Staubli VAL3: mnuMoveTargPnt.pgx

program mnuMoveTargPnt()
  local bool LbBackup
  local bool LbIsInRange
  local bool LbTestLocResult
  local joint LjHere
  local joint LjTarget
  local point LpMoveTarget
  local num nKey
begin
  //header begin
  // PROGRAM mnuMoveTargPnt()
  //
  // runs the menu to query for user to select and move to
  // Target Point
  //
  // incoming parms:  none
  // outgoing parms:  none
  // called from:  pgm mnuMotionMenu()
  //
  //  initial release KN
  //header end
  //
  // start continuous loop, end by menu command or teach pendant command
  // on user command, jump to other subroutines for action
  //
  // init booleans for menu control
  LbBackup=false
  bWorldFrameView=true
  //
  do
    //nIdxMoveTargPt=281
    call displayMessage2(nIdxMoveTargPt,nKey)
    // verify selection
    switch nKey
      // ESC key aborts & returns immediately
      case 255
        return
      break
      // Move to Target Point, F1 to change Target Frame number 1 or 2
      case 271
        nIPNumber=nIPNumber+1
        if nIPNumber==2
          nIPNumber=0
        endIf
      break
      // Move to Target Point, F2 to increment point number 0-19 in selected frame 0-1
      case 272
        if nIPNumber==0
          nIP1Number=nIP1Number+1
          if nIP1Number==20
            nIP1Number=0
          endIf
        else
          nIP2Number=nIP2Number+1
          if nIP2Number==20
            nIP2Number=0
          endIf
        endIf
      break
      // menu Move To Target Point, F5 to ADJUST RX/RY/RZ values of Target Point
      case 275
        call mnuAdjTargetPnt()
      break
      //  Move to Target Point, F6 to MOVE to currently selected IP & TP
      case 276
        // test if move to Target Point is possible
        // set up dummy loc at current location & configuration
        LjHere=jPark
        // test desired Target Point for validity
        if nIPNumber==0


          logMsg("x  "+toString(".6",tSensorTool.trsf.x))
          logMsg("y  "+toString(".6",tSensorTool.trsf.y))
          logMsg("z  "+toString(".6",tSensorTool.trsf.z))
          logMsg("rx "+toString(".6",tSensorTool.trsf.rx))
          logMsg("ry "+toString(".6",tSensorTool.trsf.ry))
          logMsg("rz "+toString(".6",tSensorTool.trsf.rz))

          logMsg("x  "+toString(".6",pIP1Point[nIP1Number].trsf.x))
          logMsg("y  "+toString(".6",pIP1Point[nIP1Number].trsf.y))
          logMsg("z  "+toString(".6",pIP1Point[nIP1Number].trsf.z))
          logMsg("rx "+toString(".6",pIP1Point[nIP1Number].trsf.rx))
          logMsg("ry "+toString(".6",pIP1Point[nIP1Number].trsf.ry))
          logMsg("rz "+toString(".6",pIP1Point[nIP1Number].trsf.rz))


          LbTestLocResult=pointToJoint(tSensorTool,LjHere,pIP1Point[nIP1Number],LjTarget)
        else
          LbTestLocResult=pointToJoint(tSensorTool,LjHere,pIP2Point[nIP2Number],LjTarget)
        endIf
        // issue error if not valid or if cannot be reached, otherwise commence move
        if LbTestLocResult==false
          LbBackup=true
          popUpMsg("IMPOSSIBLE MOVE:  Unable to reach Target Point in current arm configuration...Press OK")
          //call movTargetPoint()
        else
          LbIsInRange=isInRange(LjTarget)
          if LbIsInRange==true
            call movTargetPoint()
          else
            popUpMsg("IMPOSSIBLE MOVE:  Target Point out of reach or out of limits...Press OK")
          endIf
        endIf
      break
      // menu = Move Target Points, F7 to change displayed trsf values relative to the selected IP or World CoordSys
      // this boolean is acted upon in pgm displayMessage2()
      case 277
        if bWorldFrameView==true
          bWorldFrameView=false
        else
          bWorldFrameView=true
        endIf
      break
      //F8 to Go Back
      case 278
        LbBackup=true
      break
      // Any other key press
      default
        popUpMsg("BAD SELECTION...press OK")
      break
    endSwitch
  until (false or (LbBackup==true))
  // done
end
